(* IEC 61131-3 sources: programs/VI-54/VI-54_20171205/VI-54_20171205/Stations/Screen/LseClass170718/Class/Logic_And, 1 file *)

(* ---- Logic_And.st ---- *)
(*!
<Class
	Name               = "Logic_And"
	Revision           = "0.0"
	RealtimeTask       = "false"
	CyclicTask         = "false"
	BackgroundTask     = "false"
	Sigmatek           = "false"
	OSInterface        = "false"
	HighPriority       = "false"
	Automatic          = "false"
	UpdateMode         = "Prescan"
	SharedCommandTable = "true"
	Objectsize         = "(390,360)">
	<Channels>
		<Server Name="ClassSvr" Visualized="false" Initialize="false" WriteProtected="true" Retentive="false"/>
		<Server Name="result" Visualized="true" Remotely="true" Initialize="false" WriteProtected="true" Retentive="false" Comment="result of the calculation of operand1 - operand10"/>
		<Client Name="Logic_And_101" Required="true" Internal="true"/>
		<Client Name="Op1" Required="false" Internal="false" Comment="Operand 1"/>
		<Client Name="Op2" Required="false" Internal="false" Comment="Operand 2"/>
		<Client Name="Op3" Required="false" Internal="false" Comment="Operand 3"/>
		<Client Name="Op4" Required="false" Internal="false" Comment="Operand 4"/>
		<Client Name="Op5" Required="false" Internal="false" Comment="Operand 5"/>
	</Channels>
	<Network Name="Logic_And">
		<!-- List of Components in this network -->
		<Components>
			<Object
				Name       = "Logic_And_101"
				Class      = "Logic_And_10"
				Position   = "(210,120)"
				Visualized = "true"
				Remotely   = "true">
				<Channels>
					<Server Name="result"/>
					<Client Name="Op1"/>
					<Client Name="Op10" Value="1"/>
					<Client Name="Op2"/>
					<Client Name="Op3"/>
					<Client Name="Op4"/>
					<Client Name="Op5"/>
					<Client Name="Op6" Value="1"/>
					<Client Name="Op7" Value="1"/>
					<Client Name="Op8" Value="1"/>
					<Client Name="Op9" Value="1"/>
				</Channels>
			</Object>
		</Components>
		<Comments>
		</Comments>
		<!-- List of Connections in this network -->
		<Connections>
			<Connection Source="this.Logic_And_101" Destination="Logic_And_101.result"/>
			<Connection Source="this.result" Destination="Logic_And_101.result" Vertices="(682,270),(510,210),"/>
			<Connection Source="Logic_And_101.Op1" Destination="this.Op1" Vertices="(210,210),(38,210),"/>
			<Connection Source="Logic_And_101.Op2" Destination="this.Op2" Vertices="(210,270),(38,270),"/>
			<Connection Source="Logic_And_101.Op3" Destination="this.Op3" Vertices="(210,330),(38,330),"/>
			<Connection Source="Logic_And_101.Op4" Destination="this.Op4" Vertices="(210,390),(38,390),"/>
			<Connection Source="Logic_And_101.Op5" Destination="this.Op5" Vertices="(210,450),(38,450),"/>
		</Connections>
		<!-- Headerfiles -->
		<Options>
		</Options>
	</Network>
</Class>
*)
Logic_And : CLASS
  //Servers:
	ClassSvr 	: SvrChCmd_DINT;
	result 	: SvrCh_DINT;
  //Clients:
	Logic_And_101 	: CltChCmd_Logic_And_10;
	Op1 	: CltCh_DINT;
	Op2 	: CltCh_DINT;
	Op3 	: CltCh_DINT;
	Op4 	: CltCh_DINT;
	Op5 	: CltCh_DINT;
  //Variables:
  //Functions:

	FUNCTION VIRTUAL GLOBAL result::Read
		VAR_OUTPUT
			output (EAX) 	: DINT;
		END_VAR;
  //Tables:
	FUNCTION @STD
		VAR_OUTPUT
			ret_code	: CONFSTATES;
		END_VAR;
	FUNCTION GLOBAL TAB @CT_;
END_CLASS;

#pragma using Logic_And_10

FUNCTION VIRTUAL GLOBAL Logic_And::result::Read
	VAR_OUTPUT
		output (EAX) 	: DINT;
	END_VAR

	result := Logic_And_101.result.Read();
	output := result;

END_FUNCTION
